TYPE ST_AlertLight :
STRUCT
	Orange  : BOOL;
    Green   : BOOL;
    Red     : BOOL;
END_STRUCT
END_TYPE

(* stored: Version 1.1.0.1, ProductVersion 3.1.4024.9
   DUT ST_AlertLight: Id {c55aa9e1-d14f-4fc5-ba11-f5796180248e} *)
